DATA_BLOCK DBPOSICAO
TITLE = Titulo
{ S7_Optimized_Access := 'FALSE' }
AUTHOR : 'Caio Ribeiro'
//COMENTARIO
VERSION : 0.0
"FB_CM_AV"

BEGIN


END_DATA_BLOCK

